(* CODESYS project Stop light.project

Project tree, tasks and I/O mapping:
  Device : CODESYS Control Win V3, 3S - Smart Software Solutions GmbH, order no. 305021, version 3.5.11.40
    application Application
      libraries: Standard, * (System)
      task MainTask (cyclic, interval t#20ms, priority 1) calls PLC_PRG
      task VISU_TASK (cyclic, interval 100 ms, priority 31) calls VisuElems.Visu_Prg
      program PLC_PRG [LD]
      visualisation Visualization
  text list GlobalTextList
*)

// Device/Application/PLC_PRG
PROGRAM PLC_PRG
VAR
	start: BOOL;
	stop: BOOL;
	set: BOOL;
	green: BOOL;
	yellow: BOOL;
	red: BOOL;
	F_TRIG_0: F_TRIG;
	F_TRIG_1: F_TRIG;
	TP_0: TP;
	TP_1: TP;
	TP_2: TP;
	F_TRIG_2: F_TRIG;
	TON_0: TON;
	TON_1: TON;
	TON_2: TON;
	F_TRIG_3: F_TRIG;
	F_TRIG_4: F_TRIG;
	db: BOOL;
	TON_3: TON;
	TP_3: TP;
END_VAR

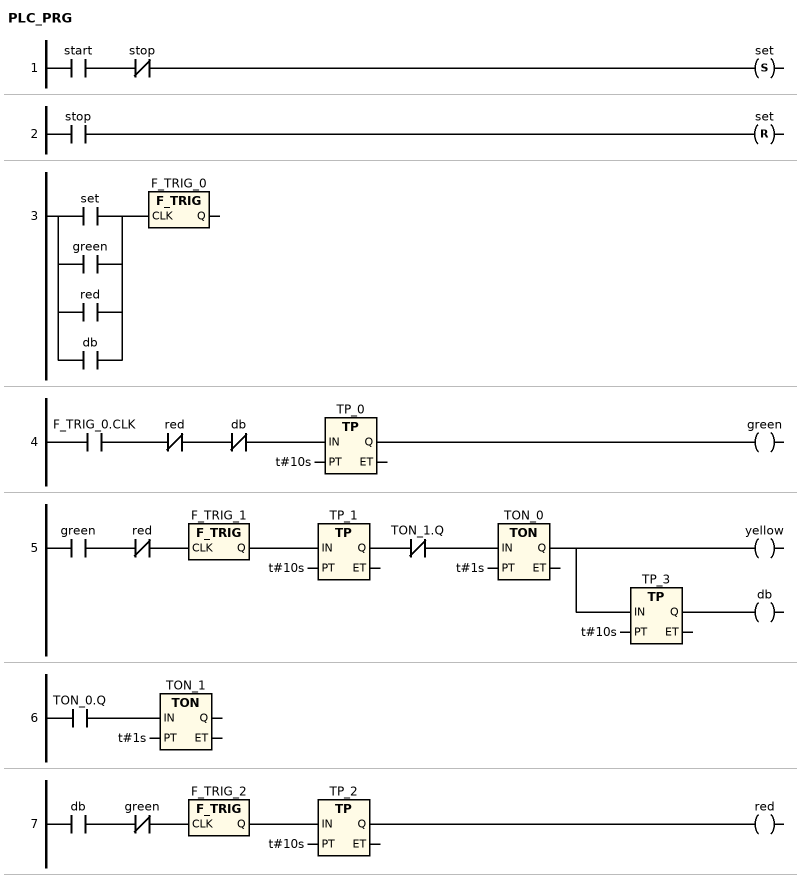
// NETWORK 1
set S= start AND NOT stop;

// NETWORK 2
set R= stop;

// NETWORK 3
F_TRIG_0(CLK := set OR green OR red OR db); // F_TRIG

// NETWORK 4
TP_0(IN := F_TRIG_0.CLK AND NOT red AND NOT db, PT := t#10s); // TP
green := TP_0.Q;

// NETWORK 5
F_TRIG_1(CLK := green AND NOT red); // F_TRIG
TP_1(IN := F_TRIG_1.Q, PT := t#10s); // TP
TON_0(IN := TP_1.Q AND NOT TON_1.Q, PT := t#1s); // TON
yellow := TON_0.Q;
TP_3(IN := TON_0.Q, PT := t#10s); // TP
db := TP_3.Q;

// NETWORK 6
TON_1(IN := TON_0.Q, PT := t#1s); // TON

// NETWORK 7
F_TRIG_2(CLK := db AND NOT green); // F_TRIG
TP_2(IN := F_TRIG_2.Q, PT := t#10s); // TP
red := TP_2.Q;

END_PROGRAM

// Device/Application/Visualization
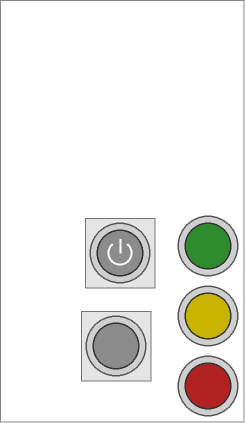
VISUALIZATION Visualization  // 245x423
    Lamp1 (173,211 70x70), variable: PLC_PRG.green, style: Lamp-Lamp1-Green
    Lamp1 (173,281 70x70), variable: PLC_PRG.yellow, style: Lamp-Lamp1-Yellow
    Lamp1 (173,351 70x70), variable: PLC_PRG.red, style: Lamp-Lamp1-Red
    PowerSwitch (85,218 70x70), variable: PLC_PRG.start, behaviour: TAP, style: Switch-PowerSwitch-Gray
    PushSwitch (81,311 70x70), variable: PLC_PRG.stop, behaviour: TAP, style: Switch-PushSwitch-Gray
END_VISUALIZATION
